INTERFACE ITF

END_INTERFACE

(* stored: Version 1.1.0.1, ProductVersion 3.1.4024.12
   Itf ITF: Id {8cfd2bbd-6ab4-459c-ac3d-5f0205344108} *)
